FUNCTION_BLOCK AssignableDigitalInputChannel implements I_DigitalInput
VAR
	digitalInput : I_DigitalInput;
END_VAR

METHOD PUBLIC ChangeDigitalInput
VAR_INPUT
	DigitalInput : I_DigitalInput;
END_VAR
IF DigitalInput <> 0 THEN
	THIS^.digitalInput := DigitalInput;
END_IF
END_METHOD

METHOD FB_init : BOOL
VAR_INPUT
	bInitRetains : BOOL; // if TRUE, the retain variables are initialized (warm start / cold start)
	bInCopyCode : BOOL;  // if TRUE, the instance afterwards gets moved into the copy code (online change)
	DigitalInput : I_DigitalInput;
END_VAR
this^.digitalInput := DigitalInput;
END_METHOD

PROPERTY PUBLIC State : BOOL
GET
State := digitalInput.State;
END_GET
END_PROPERTY

END_FUNCTION_BLOCK

(* stored: Version 1.1.0.1, ProductVersion 3.1.4024.5
   POU AssignableDigitalInputChannel: Id {eb1ad725-e598-4dff-a100-d3ce73f1e8fe}, SpecialFunc None
   Method ChangeDigitalInput: Id {15e5adc7-09e3-4e13-88e5-1bc6a0bb9f50}
   Method FB_init: Id {fd46711e-df3e-4dfb-bb82-c0f85ccda31a}
   Property State: Id {214b6653-4e33-4ee3-b621-9d0af44ceaa8}
   Get Get: Id {db02c256-e3dc-41f0-b7bb-dab9bc93ca70} *)
